% RSLogix 500 project P4_WATER_TREATMENT_SYSTEM.RSS, saved by version 8.30.00.16 %
PROJECT "UNTITLED"    % processor: Bul.1763 MicroLogix 1100 Series B %

PROGRAM FILES
  LAD 2 "MAIN"  4 rungs
  LAD 3 "IO"  7 rungs
  LAD 4 "POSITION"  6 rungs
  LAD 5 "CONTROL"  8 rungs

DATA FILES
  O0 OUTPUT  4 elements
  I1 INPUT  6 elements
  S2 STATUS  66 elements
  B3 BINARY  2 elements
  T4 TIMER  4 elements
  C5 COUNTER  1 elements
  R6 CONTROL  1 elements
  N7 INTEGER  1 elements
  F8 FLOAT  1 elements

LADDER 2 "MAIN"
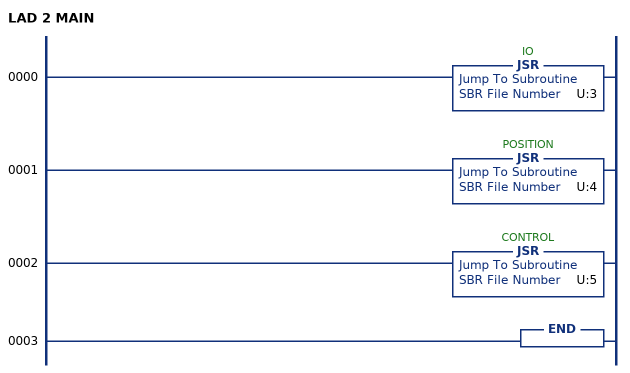
% Rung: 0 %
SOR JSR U:3 EOR
%   U:3  "IO" %
% Rung: 1 %
SOR JSR U:4 EOR
%   U:4  "POSITION" %
% Rung: 2 %
SOR JSR U:5 EOR
%   U:5  "CONTROL" %
% Rung: 3 %
SOR END EOR

LADDER 3 "IO"
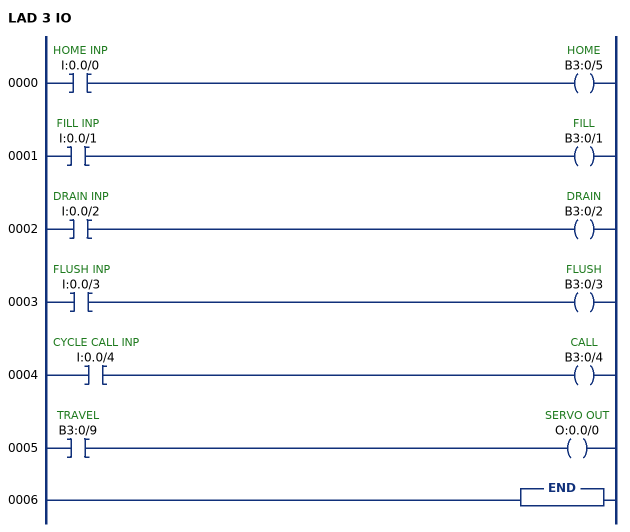
% Rung: 0 %
SOR XIC I:0.0/0 OTE B3:0/5 EOR
%   I:0.0/0  "HOME INP" %
%   B3:0/5  "HOME" %
% Rung: 1 %
SOR XIC I:0.0/1 OTE B3:0/1 EOR
%   I:0.0/1  "FILL INP" %
%   B3:0/1  "FILL" %
% Rung: 2 %
SOR XIC I:0.0/2 OTE B3:0/2 EOR
%   I:0.0/2  "DRAIN INP" %
%   B3:0/2  "DRAIN" %
% Rung: 3 %
SOR XIC I:0.0/3 OTE B3:0/3 EOR
%   I:0.0/3  "FLUSH INP" %
%   B3:0/3  "FLUSH" %
% Rung: 4 %
SOR XIC I:0.0/4 OTE B3:0/4 EOR
%   I:0.0/4  "CYCLE CALL INP" %
%   B3:0/4  "CALL" %
% Rung: 5 %
SOR XIC B3:0/9 OTE O:0.0/0 EOR
%   B3:0/9  "TRAVEL" %
%   O:0.0/0  "SERVO OUT" %
% Rung: 6 %
SOR END EOR

LADDER 4 "POSITION"
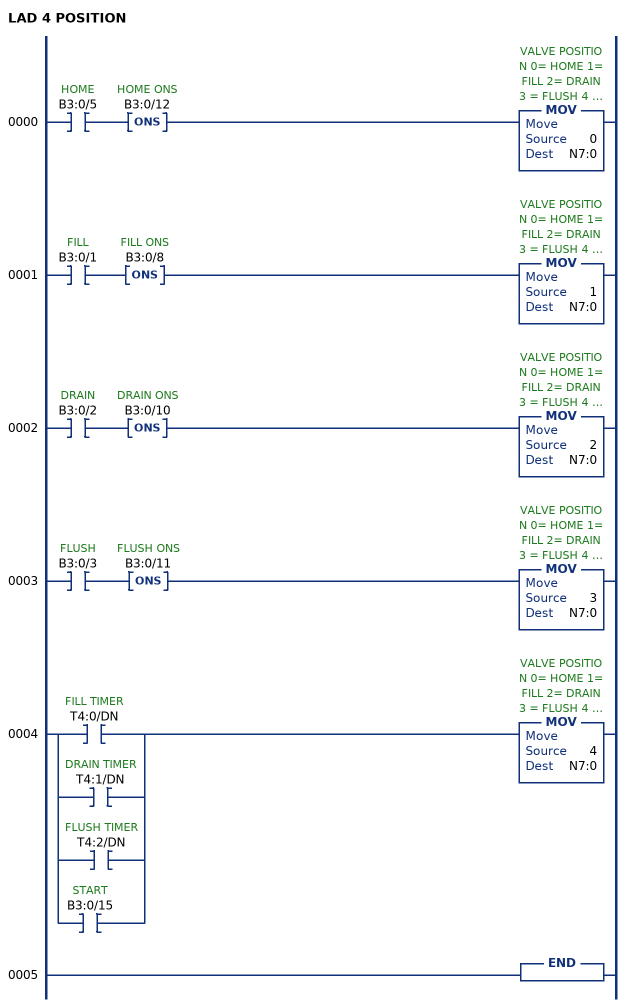
% Rung: 0 %
SOR XIC B3:0/5 ONS B3:0/12 MOV 0 N7:0 EOR
%   B3:0/5  "HOME" %
%   B3:0/12  "HOME ONS" %
%   N7:0  "VALVE POSITION 0= HOME 1= FILL 2= DRAIN 3 = FLUSH 4 = TRAVELLING" %
% Rung: 1 %
SOR XIC B3:0/1 ONS B3:0/8 MOV 1 N7:0 EOR
%   B3:0/1  "FILL" %
%   B3:0/8  "FILL ONS" %
%   N7:0  "VALVE POSITION 0= HOME 1= FILL 2= DRAIN 3 = FLUSH 4 = TRAVELLING" %
% Rung: 2 %
SOR XIC B3:0/2 ONS B3:0/10 MOV 2 N7:0 EOR
%   B3:0/2  "DRAIN" %
%   B3:0/10  "DRAIN ONS" %
%   N7:0  "VALVE POSITION 0= HOME 1= FILL 2= DRAIN 3 = FLUSH 4 = TRAVELLING" %
% Rung: 3 %
SOR XIC B3:0/3 ONS B3:0/11 MOV 3 N7:0 EOR
%   B3:0/3  "FLUSH" %
%   B3:0/11  "FLUSH ONS" %
%   N7:0  "VALVE POSITION 0= HOME 1= FILL 2= DRAIN 3 = FLUSH 4 = TRAVELLING" %
% Rung: 4 %
SOR BST XIC T4:0/DN NXB XIC T4:1/DN NXB XIC T4:2/DN NXB XIC B3:0/15 BND MOV 4 N7:0 EOR
%   T4:0  "FILL TIMER" %
%   T4:1  "DRAIN TIMER" %
%   T4:2  "FLUSH TIMER" %
%   B3:0/15  "START" %
%   N7:0  "VALVE POSITION 0= HOME 1= FILL 2= DRAIN 3 = FLUSH 4 = TRAVELLING" %
% Rung: 5 %
SOR END EOR

LADDER 5 "CONTROL"
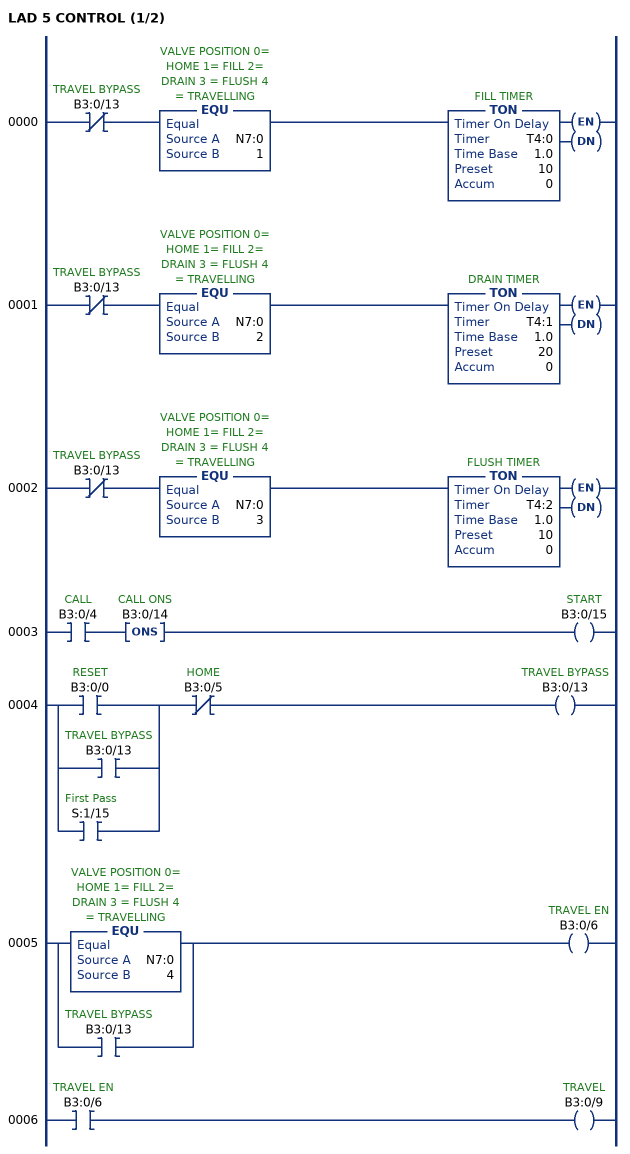
% Rung: 0 %
SOR XIO B3:0/13 EQU N7:0 1 TON T4:0 1.0 10 0 EOR
%   B3:0/13  "TRAVEL BYPASS" %
%   N7:0  "VALVE POSITION 0= HOME 1= FILL 2= DRAIN 3 = FLUSH 4 = TRAVELLING" %
%   T4:0  "FILL TIMER" %
% Rung: 1 %
SOR XIO B3:0/13 EQU N7:0 2 TON T4:1 1.0 20 0 EOR
%   B3:0/13  "TRAVEL BYPASS" %
%   N7:0  "VALVE POSITION 0= HOME 1= FILL 2= DRAIN 3 = FLUSH 4 = TRAVELLING" %
%   T4:1  "DRAIN TIMER" %
% Rung: 2 %
SOR XIO B3:0/13 EQU N7:0 3 TON T4:2 1.0 10 0 EOR
%   B3:0/13  "TRAVEL BYPASS" %
%   N7:0  "VALVE POSITION 0= HOME 1= FILL 2= DRAIN 3 = FLUSH 4 = TRAVELLING" %
%   T4:2  "FLUSH TIMER" %
% Rung: 3 %
SOR XIC B3:0/4 ONS B3:0/14 OTE B3:0/15 EOR
%   B3:0/4  "CALL" %
%   B3:0/14  "CALL ONS" %
%   B3:0/15  "START" %
% Rung: 4 %
SOR BST XIC B3:0/0 NXB XIC B3:0/13 NXB XIC S:1/15 BND XIO B3:0/5 OTE B3:0/13 EOR
%   B3:0/0  "RESET" %
%   B3:0/13  "TRAVEL BYPASS" %
%   S:1/15  "First Pass" %
%   B3:0/5  "HOME" %
% Rung: 5 %
SOR BST EQU N7:0 4 NXB XIC B3:0/13 BND OTE B3:0/6 EOR
%   N7:0  "VALVE POSITION 0= HOME 1= FILL 2= DRAIN 3 = FLUSH 4 = TRAVELLING" %
%   B3:0/13  "TRAVEL BYPASS" %
%   B3:0/6  "TRAVEL EN" %
% Rung: 6 %
SOR XIC B3:0/6 OTE B3:0/9 EOR
%   B3:0/6  "TRAVEL EN" %
%   B3:0/9  "TRAVEL" %

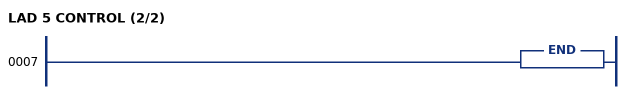
% Rung: 7 %
SOR END EOR

OTHER DOCUMENTED ADDRESSES
  F  "FF F F F FF"
  FF  "F F F FF F"
  U2  

DATA TABLE (non-zero values as saved)
DATA B3
% B3:0 % 0X0644 0X0000
DATA T4
% .PRE .ACC %
% T4:0 % 10 0
% T4:1 % 20 0
% T4:2 % 10 0
DATA N7
% N7:0 % 4
